{attribute 'qualified_only'}
VAR_GLOBAL
	// Bouton appelle ascenseur etage
	BP_EG : BOOL := FALSE;
	BP_1OG : BOOL := FALSE;
	BP_2OG : BOOL := FALSE;
	
	// Lampe 
	Lampe_EG : BOOL := FALSE;
	Lampe_1OG : BOOL := FALSE;
	Lampe_2OG : BOOL := FALSE;
	
	iEtageAppel : INT;
	iEtageActuel : INT; 
	
	MouvementAscenseur : BOOL := FALSE;
	TempsMouvementAscenseur : TON;
	
	// Ouverture Porte
	OuverturePorte : Ton;
	Lampe_Ouverture : BOOL := FALSE;
	
	// Fermeture Porte
	FermeturePorte : Ton;
	Lampe_Fermeture : Bool := False;
	
END_VAR

(* stored: Version 1.1.0.1, ProductVersion 3.1.4024.16
   GVL GVL: Id {c060a810-e345-43ad-84e2-8456f7310124} *)
